FUNCTION_BLOCK FB_Axis
VAR_INPUT
END_VAR
VAR_IN_OUT
	AxisRef	: AXIS_REF;
END_VAR
VAR_OUTPUT
	bDynamicVelocityActive	: BOOL;
	bAxisReady				: BOOL;
	bError					: BOOL;
END_VAR
VAR
	//AxisRef		: AXIS_REF;

	bReset			: BOOL;			// Rising edge triggers  reset 
	bReCalibrate	: BOOL;			// Rising edge triggers axis position reset 
	fCalPosition	: LREAL;		// The calibration position
	bPowerOn		: BOOL;			// Enable, keep high for axis enable
	bNotFastDisable	: BOOL	:= TRUE;// Used for the hard fault disable
	bDelayPowerOff	: BOOL;			// Used for controlled axis stop.
	bStopAxis		: BOOL;			// Used for controlled axis stop

	
	fbReadAxisParam		: MC_ReadParameter;	// FB to get axis max Decel
	fAxisMaxDec			: LREAL;	// The max axis Deceleration, read from the axis config

	// Motion axis functions
	McPower	: MC_Power;
	McReset	: MC_Reset;
	McHome	: MC_Home;
	
	// Edge detection 
	fbReCalibrate			: TP;
	fbExtReset				: TP;
	fbGetAxisParam			: TP;
	fbFallingExtResetQ		: F_TRIG;
	fbFallingRecalibrateQ	: F_TRIG;
	fbFallingPowerOn		: F_TRIG;
	fbRisingMcPowerStatus	: R_TRIG;
	fbRisingMcResetDone		: R_TRIG;
	fbRisingMcHomeDone		: R_TRIG;
	fbRisingStopDone		: R_TRIG;
	fbRisingHaltDone		: R_TRIG;
	fbRisingPowerON			: R_TRIG;
	
	// Distinguish between standard home and special home
	iHomeSource	: INT	:= 1; // 1 for startup home, 2 for other home function 
	
	// Dynamic velocity
	fDynamicVelo			: LREAL;
	fbFallingDynamicVelocity: F_TRIG;
	bPhase					: BOOL;
	bDvHeartBeat			: BOOL;
	bDelayHaltDisable		: BOOL;
	bBlockDynamicVelocity	: BOOL;
	McMoveVelocity_A		: MC_MoveVelocity;
	McMoveVelocity_B		: MC_MoveVelocity;
	McHalt					: MC_Halt;
	McStop					: MC_Stop;
	
	eMotionDirection		: MC_Direction;
	
	
END_VAR

// Run edge detection FB's (AXIS MANAGENEMT) 
fbRisingMcPowerStatus(CLK:=McPower.Status);
fbRisingPowerON(CLK:=bPowerOn);
fbRisingMcResetDone(CLK:=McReset.Done);
fbRisingMcHomeDone(CLK:=McHome.Done);
fbExtReset(IN:=bReset,PT:=T#2MS);
fbFallingExtResetQ(CLK:=fbExtReset.Q);
fbReCalibrate(IN:=bReCalibrate,PT:=T#2MS);
fbFallingRecalibrateQ(CLK:=fbReCalibrate.Q);
fbFallingPowerOn(CLK:=bPowerOn);
fbGetAxisParam(IN:=fbRisingMcPowerStatus.Q,PT:=T#20MS);
fbRisingStopDone(CLK:=McStop.Done);
fbRisingHaltDone(CLK:=McHalt.Done);

// Run edge detection FB's (DYNAMIC VELOCITY) 
fbFallingDynamicVelocity(CLK:=bDynamicVelocityActive);

// Delay the HALT disable to allow axis to halt when disabling dynamic velocity mode
IF(fbFallingDynamicVelocity.Q)THEN
	bDelayHaltDisable	:= TRUE;
END_IF

IF(fbRisingMcResetDone.Q) THEN
	bBlockDynamicVelocity	:= FALSE;
END_IF


IF(fbRisingStopDone.Q)THEN
	bStopAxis		:= FALSE;
	bDelayPowerOff	:= FALSE;
END_IF

IF(fbFallingPowerOn.Q)THEN
	IF(AxisRef.NcToPlc.AxisState <> 0)THEN
		bStopAxis		:= TRUE;			// trigger a controlled axis stop if the axis is disabled while running a motion
		bDelayPowerOff	:= TRUE;			// Delay the power off until the axis has come to a stop
	END_IF
END_IF

IF(fbFallingExtResetQ.Q)THEN
	bReset	:= FALSE;
END_IF

IF(fbFallingRecalibrateQ.Q)THEN
	bReCalibrate	:= FALSE;
END_IF

// Read the Max Deceleration from the axis 
fbReadAxisParam(	Axis			:= AxisRef, 
					Enable			:= fbGetAxisParam.Q,
					ParameterNumber	:= MC_AxisParameter.AxisMaximumDeceleration,
					Value			=> fAxisMaxDec);

//Check for errors 
IF(	(McPower.Error) OR 
	(McReset.Error) OR 
	(McHome.Error)	OR
	(AxisRef.NcToPlc.ErrorCode <> 0)) THEN
	
		bError := TRUE;
	
	ELSE
		bError := FALSE;
END_IF

// Run MC Power, Reset and Home Functions
McPower(	Axis			:= AxisRef,
			Enable			:= (bDelayPowerOff OR bPowerOn) AND bNotFastDisable,
			Enable_Positive	:= TRUE,
			Enable_Negative	:= TRUE,
			Override		:= 100);
			
McReset( 	Axis			:= AxisRef,
			Execute			:= (fbRisingMcPowerStatus.Q OR fbExtReset.Q OR (fbRisingPowerON.Q AND (AxisRef.NcToPlc.ErrorCode <> 0)) ));
// Home
CASE iHomeSource OF 
	1:	
		// standard start up force calibration 
		McHome( 	Axis			:= AxisRef,
					HomingMode		:= MC_HomingMode.MC_ForceCalibration,
					Execute			:= fbRisingMcResetDone.Q);
	2: 
		// recalibration function direct calibration 
		McHome( 	Axis			:= AxisRef,
					HomingMode		:= MC_HomingMode.MC_Direct,
					Position		:= fCalPosition,
					Execute			:= fbReCalibrate.Q);
	ELSE
		iHomeSource	:= 1;
END_CASE	


// Swap back to default home source when home completes
IF(fbRisingMcHomeDone.Q)THEN
	iHomeSource	:= 1;
END_IF	

// Set the output axis ready flag					
IF(bPowerOn AND fbRisingMcHomeDone.Q AND NOT(bError))THEN
	bAxisReady	:= TRUE;
END_IF		

// Reset the output axis ready flag 
IF(NOT(bPowerOn) OR bError)THEN
	bAxisReady	:= FALSE;	
END_IF



// Dynamic Velocity Implementation
IF(bDynamicVelocityActive AND NOT(bBlockDynamicVelocity)) THEN
	
	bPhase	:= NOT(bPhase);	// Phase alternator to allow continuous target velocity updates
	
	McMoveVelocity_A( 	Axis			:= AxisRef,
						Execute			:= (bPhase AND (fDynamicVelo <> 0) AND bPowerOn),
						Direction		:= eMotionDirection,
						Velocity		:= ABS(fDynamicVelo));
	
	McMoveVelocity_B( 	Axis			:= AxisRef,
						Execute			:= (NOT(bPhase) AND (fDynamicVelo <> 0) AND bPowerOn),
						Direction		:= eMotionDirection,
						Velocity		:= ABS(fDynamicVelo));
	
	
	// Run a heartbeat to disablle dynamic velocity as soon as the user stops updating it					
	IF(NOT(bDvHeartBeat))THEN
		bDynamicVelocityActive	:= FALSE;
	END_IF
	
	// Reset the dynamic velocity active state
	bDvHeartBeat	:= FALSE;
	
						
END_IF 

IF(bDynamicVelocityActive OR bDelayHaltDisable) THEN
	// This is used for dynamic velocity mode 
	McHalt			(	Axis			:= AxisRef,
						Deceleration	:= fAxisMaxDec,
						Execute			:= ((fDynamicVelo = 0) AND bPowerOn) OR fbFallingDynamicVelocity.Q);
	
	// reset bDelay halt disable when the halt function completes 
	IF(fbRisingHaltDone.Q)THEN
		bDelayHaltDisable	:= FALSE;
	END_IF
						
END_IF

// Implement a max dec controller axis Stop if the axis is disabled while running a motion
McStop			(	Axis			:= AxisRef,
					Deceleration	:= fAxisMaxDec,
					Execute			:= bStopAxis);

METHOD Disable : BOOL // Disbales the axis after stopping the axis as fast as possible , graceful stop 
VAR_INPUT
END_VAR
THIS^.bPowerOn				:= FALSE;
END_METHOD

METHOD DynamicVelocity : BOOL
VAR_INPUT
	fVelocity	: LREAL;
END_VAR
IF(THIS^.bAxisReady) THEN 
	IF(NOT(bDynamicVelocityActive)) THEN THIS^.bDynamicVelocityActive := TRUE; END_IF // Assert the dynamic velocity active flag 
	THIS^.bDvHeartBeat 			:= TRUE;		// Run the dynamic velocity active heartbeat 
	THIS^.fDynamicVelo			:= fVelocity;	// Update the target velocity
	IF(fVelocity > 0)THEN
		THIS^.eMotionDirection	:= MC_Direction.MC_Positive_Direction;
	ELSE
		THIS^.eMotionDirection	:= MC_Direction.MC_Negative_Direction;
	END_IF
END_IF
END_METHOD

METHOD Enable : BOOL
VAR_INPUT
END_VAR
THIS^.bPowerOn					:= TRUE;
THIS^.bNotFastDisable			:= TRUE;
THIS^.bDynamicVelocityActive	:= FALSE;
END_METHOD

METHOD FastDisable : BOOL	// Disbales the axis immediately, if moving will result in a fault
VAR_INPUT
END_VAR
THIS^.bNotFastDisable	:= FALSE;
END_METHOD

METHOD Reset : BOOL
VAR_INPUT
END_VAR
THIS^.bReset					:= TRUE;
THIS^.bDynamicVelocityActive	:= FALSE;
END_METHOD

METHOD ResetPosition : BOOL
VAR_INPUT
	fPosition	: LREAL; 	// Calibration axis position 
END_VAR
bReCalibrate		:= TRUE;
fCalPosition		:= fPosition;
THIS^.iHomeSource	:= 2;
END_METHOD

METHOD Stop : BOOL
VAR_INPUT
END_VAR
THIS^.bStopAxis					:= TRUE;
THIS^.bBlockDynamicVelocity		:= TRUE;
END_METHOD

END_FUNCTION_BLOCK

(* stored: Version 1.1.0.1, ProductVersion 3.1.4024.4
   POU FB_Axis: Id {a7595f3e-0067-4b32-bbdd-698f783f05a3}, SpecialFunc None
   Method Disable: Id {294c13ee-21ce-4669-8734-54682c297951}
   Method DynamicVelocity: Id {c8e45f90-edb1-4f0d-aa08-b06cd416349c}
   Method Enable: Id {232ab3d2-1318-44a2-aacc-890807d715fd}
   Method FastDisable: Id {f44f1294-a5cd-4c09-b324-34aea0f4be2d}
   Method Reset: Id {43b0f955-aab6-4669-99ff-7f3fb207acc2}
   Method ResetPosition: Id {09d8a13e-bdc0-40cc-a7d2-f240d9fe5cc4}
   Method Stop: Id {16bc3a7d-5d9e-48a3-931b-b5dcc481fa28} *)
